// TIA Portal project "thuoc" (V16)

(* hardware
DEVICE "S7-1200 station_1"  S7-1200 Station
   slot 0: "Rack_0"  S7-1200 Rack  Rack  V1.0
   slot 1: "PLC_1"  CPU 1212C DC/DC/Rly  6ES7 212-1HE40-0XB0  V4.4
*)

// ===== PLC "PLC_1"  CPU 1212C DC/DC/Rly =====

VAR_GLOBAL   // PLC tag table "Default tag table"
   "Tag_1" AT %M0.0 : Bool;
   "Tag_2" AT %M0.1 : Bool;
   "Tag_3" AT %M0.2 : Bool;
   "Tag_4" AT %M10.0 : Bool;
   "Tag_5" AT %M100.0 : Bool;
   "Tag_6" AT %M100.1 : Bool;
   "System_Byte" AT %MB1 : Byte;
   "FirstScan" AT %M1.0 : Bool;
   "DiagStatusUpdate" AT %M1.1 : Bool;
   "AlwaysTRUE" AT %M1.2 : Bool;
   "AlwaysFALSE" AT %M1.3 : Bool;
   "System_Byte(1)" AT %MB1 : Byte;
END_VAR

VAR_GLOBAL   // PLC tag table "Tag table_2"
   "den" AT %Q0.0 : Bool;
   "bang tai" AT %Q0.1 : Bool;
   "led xanh" AT %Q0.2 : Bool;
   "led do" AT %Q0.3 : Bool;
   "xi lanh" AT %Q0.4 : Bool;
END_VAR

VAR_GLOBAL   // PLC tag table "Tag table_1"
   "btn_xanh" AT %I0.0 : Bool;
   "btn_den" AT %I0.1 : Bool;
   "emry" AT %I0.3 : Bool;
   "switch" AT %I0.2 : Bool;
   "cam bien" AT %I0.4 : Bool;
END_VAR

DATA_BLOCK "Data_block_1"   // DB1
{ S7_Optimized_Access := 'FALSE' }
VERSION : 0.1
   VAR
      Result_NG : Bool;
      Sensor_Trigger : Bool;
      Conveyor_Run : Bool;
      System_Active : Bool;
      Result_OK : Bool;
      Camera_Online : Bool;
      num_ok : Int;
      num_ng : Int;
      num_total : Int;
      product_id : Int;
      vien_ok : Int;
      vien_ng : Int;
      vi_ok : Int;
      vi_ng : Int;
      Remote_Control : Int := 1;
   END_VAR
BEGIN
END_DATA_BLOCK

DATA_BLOCK "DB10"   // DB2
{ S7_Optimized_Access := 'FALSE' }
VERSION : 0.1
   VAR
      Tong_So_Thuoc : Int;
      Thuoc_OK : Int;
      Thuoc_NG : Int;
      Trang_Thai_He_Thong : Int;
      Web_Product_ID : Int;
      Web_CMD : Int;
   END_VAR
BEGIN
END_DATA_BLOCK

DATA_BLOCK "DB11_Modbus"   // DB5
{ S7_Optimized_Access := 'FALSE' }
VERSION : 0.1
   VAR
      Ket_Noi : TCON_IP_v4;
   END_VAR
BEGIN
   Ket_Noi.InterfaceId := 64;
   Ket_Noi.ID := 2;
   Ket_Noi.ConnectionType := 11;
   Ket_Noi.ActiveEstablished := false;
   Ket_Noi.LocalPort := 502;
END_DATA_BLOCK

ORGANIZATION_BLOCK "Main"   // OB1, LAD, ProgramCycle
TITLE = "Main Program Sweep (Cycle)"
{ S7_Optimized_Access := 'TRUE' }
VERSION : 0.1
   VAR_INPUT
      Initial_Call : Bool;   // Initial call of this OB
      Remanence : Bool;   // =True, if remanent data are available
   END_VAR
   VAR_TEMP   // added for the SCL form of the ladder/FBD networks
      _w1 : Bool;
   END_VAR
BEGIN

REGION Network 1
   // dieu khien bang tay , tu xa tren web va reset tung loai thuoc
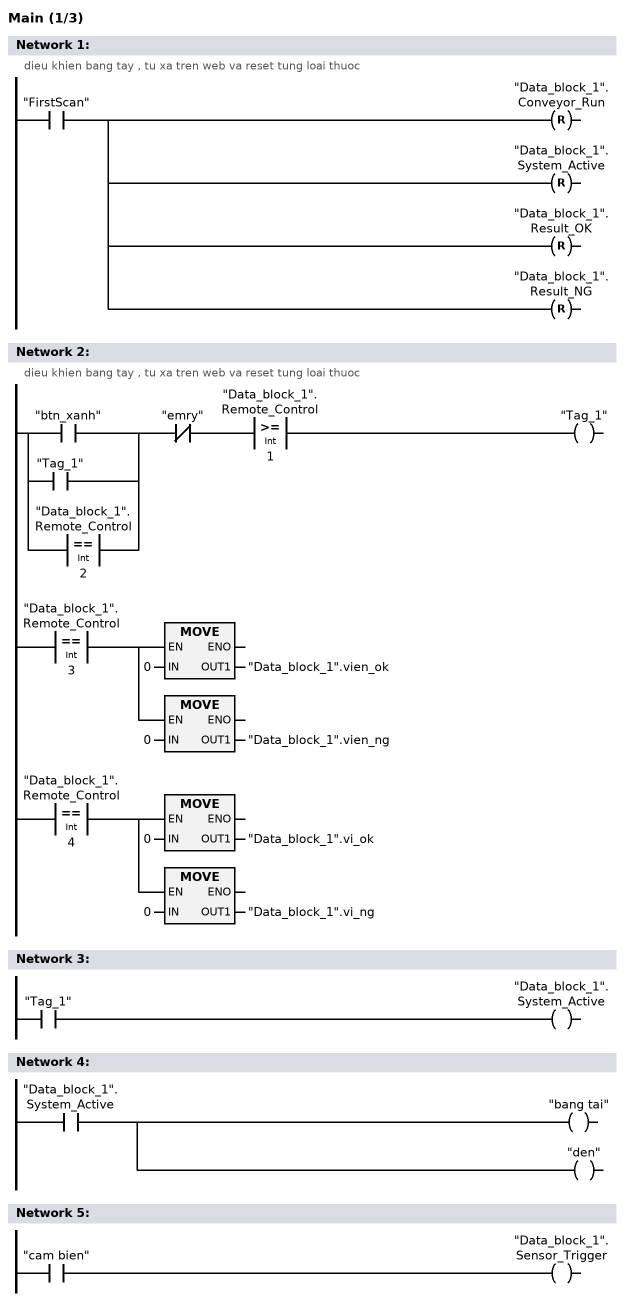
   RUNG wire#powerrail
      Contact( "FirstScan" )
      wire#w1
      R_Coil( "Data_block_1".Conveyor_Run )
   END_RUNG
   RUNG wire#w1
      R_Coil( "Data_block_1".System_Active )
   END_RUNG
   RUNG wire#w1
      R_Coil( "Data_block_1".Result_OK )
   END_RUNG
   RUNG wire#w1
      R_Coil( "Data_block_1".Result_NG )
   END_RUNG
   // the same network as SCL:
   IF "FirstScan" THEN
       "Data_block_1".Conveyor_Run := FALSE;
       "Data_block_1".System_Active := FALSE;
       "Data_block_1".Result_OK := FALSE;
       "Data_block_1".Result_NG := FALSE;
   END_IF;
END_REGION

REGION Network 2
   // dieu khien bang tay , tu xa tren web va reset tung loai thuoc
   RUNG wire#powerrail
      Contact( "btn_xanh" )
      wire#w1
      I_Contact( "emry" )
      { S7_Templates := "SrcType := Int" } GE_Contact(in1 := "Data_block_1".Remote_Control, in2 := 1)
      Coil( "Tag_1" )
   END_RUNG
   RUNG wire#powerrail
      Contact( "Tag_1" )
   END_RUNG wire#w1
   RUNG wire#powerrail
      { S7_Templates := "SrcType := Int" } EQ_Contact(in1 := "Data_block_1".Remote_Control, in2 := 2)
   END_RUNG wire#w1
   RUNG wire#powerrail
      { S7_Templates := "SrcType := Int" } EQ_Contact(in1 := "Data_block_1".Remote_Control, in2 := 3)
      wire#w2
      Move(in := 0, out1 => "Data_block_1".vien_ok)
   END_RUNG
   RUNG wire#w2
      Move(in := 0, out1 => "Data_block_1".vien_ng)
   END_RUNG
   RUNG wire#powerrail
      { S7_Templates := "SrcType := Int" } EQ_Contact(in1 := "Data_block_1".Remote_Control, in2 := 4)
      wire#w3
      Move(in := 0, out1 => "Data_block_1".vi_ok)
   END_RUNG
   RUNG wire#w3
      Move(in := 0, out1 => "Data_block_1".vi_ng)
   END_RUNG
   // the same network as SCL:
   "Tag_1" := ("btn_xanh" OR "Tag_1" OR ("Data_block_1".Remote_Control = 2)) AND NOT "emry" AND ("Data_block_1".Remote_Control >= 1);
   IF "Data_block_1".Remote_Control = 3 THEN
       "Data_block_1".vien_ok := 0;
       "Data_block_1".vien_ng := 0;
   END_IF;
   IF "Data_block_1".Remote_Control = 4 THEN
       "Data_block_1".vi_ok := 0;
       "Data_block_1".vi_ng := 0;
   END_IF;
END_REGION

REGION Network 3
   RUNG wire#powerrail
      Contact( "Tag_1" )
      Coil( "Data_block_1".System_Active )
   END_RUNG
   // the same network as SCL:
   "Data_block_1".System_Active := "Tag_1";
END_REGION

REGION Network 4
   RUNG wire#powerrail
      Contact( "Data_block_1".System_Active )
      wire#w1
      Coil( "bang tai" )
   END_RUNG
   RUNG wire#w1
      Coil( "den" )
   END_RUNG
   // the same network as SCL:
   "bang tai" := "Data_block_1".System_Active;
   "den" := "Data_block_1".System_Active;
END_REGION

REGION Network 5
   RUNG wire#powerrail
      Contact( "cam bien" )
      Coil( "Data_block_1".Sensor_Trigger )
   END_RUNG
   // the same network as SCL:
   "Data_block_1".Sensor_Trigger := "cam bien";
END_REGION

REGION Network 6
   // dk tam de xi lanh day k cam bien
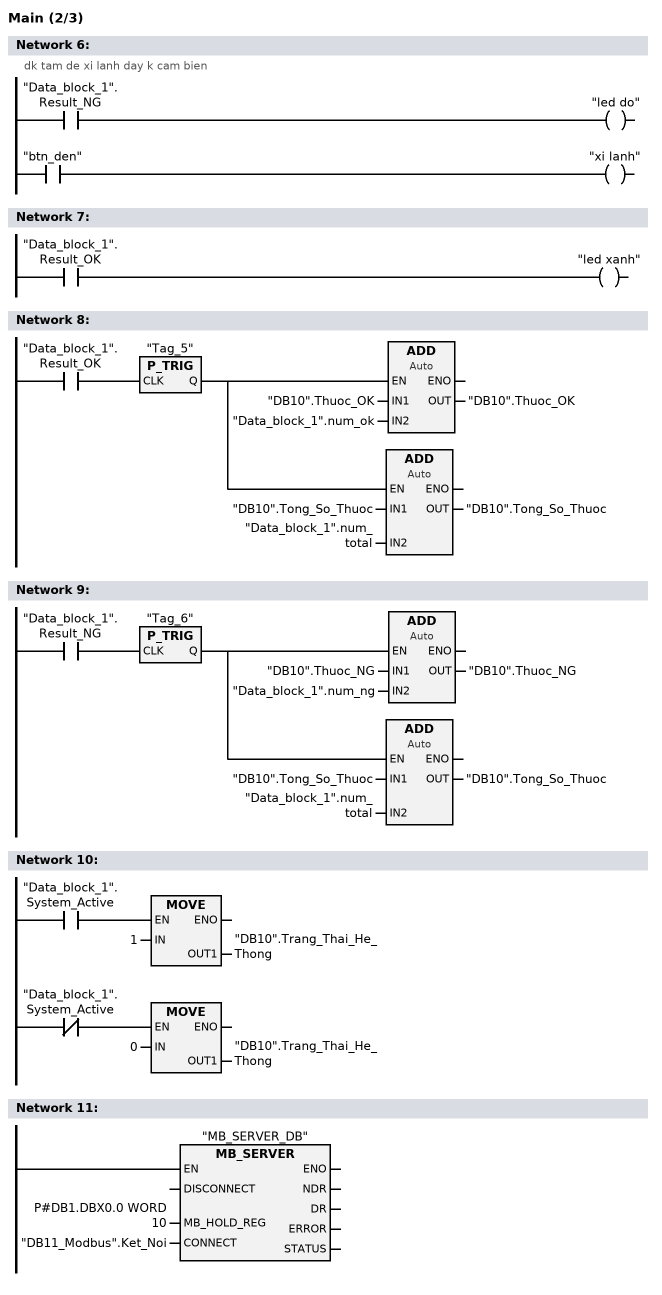
   RUNG wire#powerrail
      Contact( "Data_block_1".Result_NG )
      Coil( "led do" )
   END_RUNG
   RUNG wire#powerrail
      Contact( "btn_den" )
      Coil( "xi lanh" )
   END_RUNG
   // the same network as SCL:
   "led do" := "Data_block_1".Result_NG;
   "xi lanh" := "btn_den";
END_REGION

REGION Network 7
   RUNG wire#powerrail
      Contact( "Data_block_1".Result_OK )
      Coil( "led xanh" )
   END_RUNG
   // the same network as SCL:
   "led xanh" := "Data_block_1".Result_OK;
END_REGION

REGION Network 8
   RUNG wire#powerrail
      Contact( "Data_block_1".Result_OK )
      P_Trig( "Tag_5" )
      wire#w1
      Add(in1 := "DB10".Thuoc_OK, in2 := "Data_block_1".num_ok, out => "DB10".Thuoc_OK)
   END_RUNG
   RUNG wire#w1
      Add(in1 := "DB10".Tong_So_Thuoc, in2 := "Data_block_1".num_total, out => "DB10".Tong_So_Thuoc)
   END_RUNG
   // the same network as SCL:
   #_w1 := "Data_block_1".Result_OK AND NOT "Tag_5";   // rising edge
   "Tag_5" := "Data_block_1".Result_OK;
   IF #_w1 THEN
       "DB10".Thuoc_OK := "DB10".Thuoc_OK + "Data_block_1".num_ok;
       "DB10".Tong_So_Thuoc := "DB10".Tong_So_Thuoc + "Data_block_1".num_total;
   END_IF;
END_REGION

REGION Network 9
   RUNG wire#powerrail
      Contact( "Data_block_1".Result_NG )
      P_Trig( "Tag_6" )
      wire#w1
      Add(in1 := "DB10".Thuoc_NG, in2 := "Data_block_1".num_ng, out => "DB10".Thuoc_NG)
   END_RUNG
   RUNG wire#w1
      Add(in1 := "DB10".Tong_So_Thuoc, in2 := "Data_block_1".num_total, out => "DB10".Tong_So_Thuoc)
   END_RUNG
   // the same network as SCL:
   #_w1 := "Data_block_1".Result_NG AND NOT "Tag_6";   // rising edge
   "Tag_6" := "Data_block_1".Result_NG;
   IF #_w1 THEN
       "DB10".Thuoc_NG := "DB10".Thuoc_NG + "Data_block_1".num_ng;
       "DB10".Tong_So_Thuoc := "DB10".Tong_So_Thuoc + "Data_block_1".num_total;
   END_IF;
END_REGION

REGION Network 10
   RUNG wire#powerrail
      Contact( "Data_block_1".System_Active )
      Move(in := 1, out1 => "DB10".Trang_Thai_He_Thong)
   END_RUNG
   RUNG wire#powerrail
      I_Contact( "Data_block_1".System_Active )
      Move(in := 0, out1 => "DB10".Trang_Thai_He_Thong)
   END_RUNG
   // the same network as SCL:
   IF "Data_block_1".System_Active THEN "DB10".Trang_Thai_He_Thong := 1; END_IF;
   IF NOT "Data_block_1".System_Active THEN "DB10".Trang_Thai_He_Thong := 0; END_IF;
END_REGION

REGION Network 11
   "MB_SERVER_DB"(MB_HOLD_REG := P#DB1.DBX0.0 WORD 10, CONNECT := "DB11_Modbus".Ket_Noi);   // MB_SERVER
END_REGION

REGION Network 12
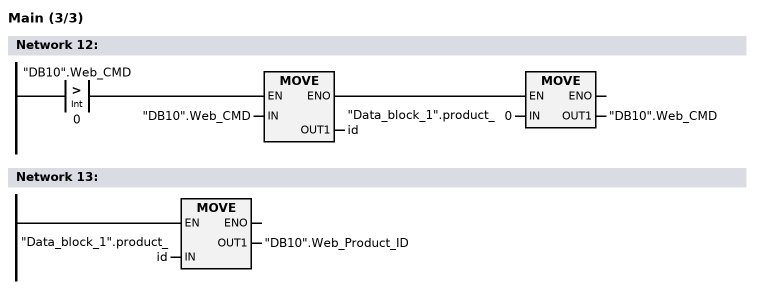
   RUNG wire#powerrail
      { S7_Templates := "SrcType := Int" } GT_Contact(in1 := "DB10".Web_CMD, in2 := 0)
      Move(in := "DB10".Web_CMD, out1 => "Data_block_1".product_id)
      Move(in := 0, out1 => "DB10".Web_CMD)
   END_RUNG
   // the same network as SCL:
   IF "DB10".Web_CMD > 0 THEN
       "Data_block_1".product_id := "DB10".Web_CMD;
       "DB10".Web_CMD := 0;
   END_IF;
END_REGION

REGION Network 13
   RUNG wire#powerrail
      Move(in := "Data_block_1".product_id, out1 => "DB10".Web_Product_ID)
   END_RUNG
   // the same network as SCL:
   "DB10".Web_Product_ID := "Data_block_1".product_id;
END_REGION
END_ORGANIZATION_BLOCK